PROGRAM ProgramPLC
VAR
	a: WORD;
END_VAR

a:=a+1;
IF A > 9999 THEN	
	A :=0;
END_IF

(*Configuracion de los Modulos*)
pConfig();

(*Activar Funciones*)
pFuctions();

(*Activar salidas*)
pActvOutputs();

(*============================================================================
21/06/2022 EDU inici comentaris*)

END_PROGRAM

(* stored: Version 1.1.0.1, ProductVersion 3.1.4024.10
   POU ProgramPLC: Id {485eb957-f196-4400-8af7-77641c0ae79e}, SpecialFunc None *)
